# EPICS autosave request: apps/myaDataApp/Db/wireScanData.req
#
# EPICS PVs for integrating scan data with the Mya archiver
#
#
# Notes:
#   [Macros]
#   P - prefix (ex. HPS_SVT:SCAN:)
#   R - prefix
#
#   [autosave]
#   Requires autosave to prevent false archived data.
#   Restore pass0.
#
# Author: Wesley Moore
# Date:   Mar 2015
#

$(P)$(R)mean_horiz
$(P)$(R)mean_stereo
$(P)$(R)x_offset
$(P)$(R)y_offset
$(P)$(R)peak_horiz
$(P)$(R)peak_stereo
$(P)$(R)sigma_y
